PROGRAM MAIN
VAR
END_VAR

(* 
	GOF 		Ensure a class only has one instance, and provide a global point of access to it.
*)
P_Singleton();

END_PROGRAM

(* stored: Version 1.1.0.1, ProductVersion 3.1.4024.12
   POU MAIN: Id {943b8dd8-8cec-4e6a-b705-026f7d031610}, SpecialFunc None *)
